TEXTLIST TextListPPMStates
  0 = 'Unknown'
  1 = 'Out'
  2 = 'Power Meter'
  3 = 'Polished Yag'
  4 = 'Frosted Yag'
   = ''
END_TEXTLIST

(* stored: Version 1.1.0.1, ProductVersion 3.1.4022.18
   TextList TextListPPMStates: Id {e6fba008-7877-4954-b26e-3d90f8256bb6} *)
